Universal Robots PolyScope program: Search.urp

ProgramRoot directory=/home/ur/ursim-3.1/programs/Support site; kinematics=(a=[0, -0.425, -0.39225, 0, 0, 0], d=[0.08916, 0, 0, 0.10915, 0.09465, 0.0823], alpha=[1.5708, 0, 0, 1.5708, -1.5708, 0], deltaTheta=[0, 0, 0, 0, 0, 0], status=notInitialized); lastSavedInVersion=(project__name=Polyscope, major__version=3, minor__version=1, svn__revision=18024, build__date=Jul 07 2015, 15:18:49); name=Search; programVersion=(project__name=Polyscope, major__version=3, minor__version=1, svn__revision=17195, build__date=Mar 11 2015, 13:02:28); robotEnvironmentFileName=default; serialNumberRobot=2015350001
  MainProgram cartesianAcceleration=1.2; cartesianSpeed=0.25; jointAcceleration=1.3962634015954636; jointSpeed=1.0471975511965976; sharedProcessMoveBlendRadius=0.025; motionType=JOINT_SPACE
    If checkConditionInSeperateThread=true; expr=ExpressionIONode≟ False; type=IF_NODE
      Move cartesianAcceleration=1.2; cartesianSpeed=0.25; jointAcceleration=1.3962634015954636; jointSpeed=1.0471975511965976; sharedProcessMoveBlendRadius=0.025; motionType=CARTESIAN_SPACE
        Waypoint blendRadius=0.05; cartesianAcceleration=1.2; cartesianSpeed=0.25; jointAcceleration=1.3962634015954636; jointSpeed=1.0471975511965976; nextMotionTime=2.0; stoppoint=true; useSharedBlendParameter=true; useSharedParameters=true; position=TCP in base x=-120 y=-400 z=0 mm, rx=0 ry=3.14 rz=0 rad; joints [-91.567, -118.987, -135.861, -15.154, 90.091, -1.567] deg; positionType=RELATIVE_POSITION; waypointPoseInFeatureCoordinates=(pos=(x=-0.11999996281371052, y=-0.400000035683787, z=2.1088057308425744E-8), rot=(x=3.0935149440374135E-7, y=3.139999985893489, z=-6.686739026337127E-7)); name=Search_Function; relativeFromJointPositionVector=(joint=[-1.59814, -1.66278, -2.29236, -0.7573, 1.57239, -0.02734], isUndefined=false); relativeFromToolAxisAngle=(x=3.0964941486526905E-7, y=3.1399999793753346, z=-2.9449666667450554E-7); relativeFromToolPosition=(x=-0.11999996164714996, y=-0.39999999194384533, z=0.14500004732549338)
    If type=ELSE_NODE
      Move cartesianAcceleration=1.2; cartesianSpeed=0.25; jointAcceleration=1.3962634015954636; jointSpeed=1.0471975511965976; sharedProcessMoveBlendRadius=0.025; motionType=CARTESIAN_SPACE
        Waypoint blendRadius=0.05; cartesianAcceleration=1.2; cartesianSpeed=0.25; jointAcceleration=1.3962634015954636; jointSpeed=1.0471975511965976; nextMotionTime=2.0; stoppoint=true; useSharedBlendParameter=true; useSharedParameters=true; outputFlangePose=(pos=(x=-0.12011316349511432, y=-0.4317629397815833, z=0.33440045381825007), rot=(x=-0.0012209830283371023, y=3.116276481240665, z=0.038891916168164946)); position=TCP in base x=-120.113 y=-431.763 z=334.4 mm, rx=-0.0012 ry=3.1163 rz=0.0389 rad; joints [-91.713, -84.826, -108.941, -77.706, 91.393, -1.776] deg; positionType=FIXED_POSITION; waypointPoseInFeatureCoordinates=(pos=(x=-0.12011316299633705, y=-0.4317629218220435, z=0.33440041081305716), rot=(x=-0.0012209830284087941, y=3.116276481240896, z=0.03889191616813282)); name=Else_do
